TYPE DUT_STRUCT_C000009_PROD :
STRUCT
	sCellName			:STRING := 'C000009';
	sIpAddress			:STRING := '10.38.191.60';
	sAmsNetId			:STRING := '10.38.191.60.1.1';
	sOpcUaURL			:STRING := 'opc.tcp://10.38.191.60:4840';
	sUhfRfidOpcUaURL	:STRING := 'opc.tcp://10.38.190.132:4840';
	sHfRfidOpcUaURL		:STRING := 'opc.tcp://10.38.191.66:4840';
	sStation1			:STRING := 'S000004';
	sLastingPC			:STRING := '10.38.191.65';
END_STRUCT
END_TYPE

(* stored: Version 1.1.0.1, ProductVersion 3.1.4024.6
   DUT DUT_STRUCT_C000009_PROD: Id {53d881ee-041d-41e1-a09b-0d09dbd8daac} *)
